INTERFACE I_Drive

METHOD M_Home : BOOL
VAR_INPUT
END_VAR
END_METHOD

METHOD M_MoveAbs : BOOL
VAR_INPUT
    fPosition : LREAL; // Target position in mm or degrees
    fVelocity : LREAL; // Speed for this move
END_VAR
END_METHOD

METHOD M_MoveVelocity : BOOL
VAR_INPUT
    fVelocity   : LREAL;         // Target speed in mm/s
    nDirection  : MC_Direction;  // 1 = Positive, 2 = Negative, 3 = Current
END_VAR
END_METHOD

METHOD M_Reset : BOOL
VAR_INPUT
END_VAR
END_METHOD

METHOD M_Stop : BOOL
VAR_INPUT
END_VAR
END_METHOD

PROPERTY P_Axis : REFERENCE TO AXIS_REF
GET
END_GET
END_PROPERTY

PROPERTY P_Busy : BOOL
GET
END_GET
END_PROPERTY

PROPERTY P_Enabled : BOOL
GET
END_GET
SET
END_SET
END_PROPERTY

PROPERTY P_Error : BOOL
GET
END_GET
END_PROPERTY

PROPERTY P_Ready : BOOL
GET
END_GET
END_PROPERTY

END_INTERFACE

(* stored: Version 1.1.0.1
   Itf I_Drive: Id {bac1fedb-add2-4ee9-b6e6-a090fe2bb612}
   Method M_Home: Id {81864300-7c80-4e81-8d44-3b6b80edf1a1}
   Method M_MoveAbs: Id {dd77af82-b0a4-48da-a076-c4140e59b2e0}
   Method M_MoveVelocity: Id {96debd5f-4fc8-450d-b944-51a9099b3993}
   Method M_Reset: Id {c038a8fe-c703-45b7-a21c-6003194c8028}
   Method M_Stop: Id {d0446528-b54f-429e-9648-2847bcd2375c}
   Property P_Axis: Id {eda4508a-df38-42ba-8ca4-a7131309c777}
   Get Get: Id {ee71f141-6459-44ab-b94c-8cc5508c2bab}
   Property P_Busy: Id {4f7370ed-5031-445d-b4e4-3dfd735989e5}
   Get Get: Id {9c69d565-c6d0-4e09-9883-0f4cdb58c5be}
   Property P_Enabled: Id {df317725-f34a-4c84-b136-bfef60668404}
   Get Get: Id {31f363a8-2f4c-425c-b929-024e77eb7c25}
   Set Set: Id {1aeb234b-677e-4bdd-bdd6-9796b2ebfe8d}
   Property P_Error: Id {66187986-7ec2-4899-8ce5-d4eef857d2e5}
   Get Get: Id {6336c5d8-1650-487f-91d5-8116a0bd4284}
   Property P_Ready: Id {fb1f186b-f398-43e4-a159-720f403e7051}
   Get Get: Id {59af60eb-274d-4b58-859e-627e317109bb} *)
